FUNCTION_BLOCK FB_Batch
VAR_INPUT
	i_bOpen						:BOOL; 
	i_bClose					:BOOL; 
	i_sBatchID					:STRING; 
	i_sBatchSubID				:STRING;
	i_sRecipe					:STRING;
	i_sProductName				:STRING;
	i_bCreateReport				:BOOL;
	i_bSendReport				:BOOL;
END_VAR
VAR_IN_OUT
	q_stParams					:ST_Batch;
	q_stLastBatch				:ST_Batch;
END_VAR
VAR_OUTPUT
	q_bBusy						:BOOL;	
	q_bOpened					:BOOL:=FALSE; 
	q_bClosed					:BOOL:=FALSE; 		
END_VAR

VAR
	tDelayCreateReport			:TON;
	tDelaySendReport			:TON;
END_VAR	

VAR PERSISTENT
	iStep						:INT;
	sUserOpened					:STRING;
END_VAR

tDelayCreateReport(IN:=(iStep=200),PT:=T#3S);
tDelaySendReport(IN:=(iStep=300),PT:=T#3S);

CASE iStep OF

	0: 
		MEMSET(ADR(q_stParams),0,SIZEOF(q_stParams));
		IF i_bOpen THEN
			iStep:=50;
		END_IF
		
	50:
		IF i_sBatchSubID <> '0' THEN
			q_stParams.sBatchNumber:=CONCAT(i_sBatchID,'-');
			q_stParams.sBatchNumber:=CONCAT(q_stParams.sBatchNumber,i_sBatchSubID);
		ELSE
			q_stParams.sBatchNumber:=i_sBatchID;
		END_IF
		q_stParams.sRecipeName:=i_sRecipe;
		q_stParams.sProductName:=i_sProductName;
		q_stParams.sUser:=GV.sUserLogged;
		q_stParams.sStarted:=GV.stTime.sDateTime;
		sUserOpened:=GV.sUserLogged;
		iStep:=100;
			
	100:
		q_stParams.sUser:=sUserOpened;
		IF i_bClose THEN
			q_stParams.sFinished:=GV.stTime.sDateTime;
			q_stLastBatch:=q_stParams;
			iStep:=200;
		END_IF
		
	200:
		IF tDelayCreateReport.Q AND NOT i_bCreateReport THEN
			iStep:=300;
		END_IF
	300:
		IF tDelaySendReport.Q AND NOT i_bSendReport THEN
			iStep:=1000;
		END_IF
		
	1000:
		iStep:=0;	
END_CASE

q_bBusy:=iStep<>0;
q_bOpened:=iStep=100;
q_bClosed:=iStep>100;

END_FUNCTION_BLOCK

(* stored: Version 1.1.0.1
   POU FB_Batch: Id {fe7fd090-901c-413f-80f9-8b402fd3e9cb}, SpecialFunc None *)
